# EPICS substitutions: iocBoot/InstekPSP/Omega.substitutions
file "$(IP)/ipApp/Db/Instek.db" { pattern
{P,          R,       PORT,    LOPR,  HOPR,   PREC, EGU,   SCAN,        CONFIG_SCAN}
{13Instek:, Omega1,  serial1,    0,  2000,   1,    PSI,   ".5 second", "5 second"}
}
